PROGRAM prgMotoman
VAR
	pReal	: POINTER TO REAL;
	rVal	: REAL;
	
	pInt	: POINTER TO INT;
	iVal	: INT;
	
	fbsin	: BASIC.GEN_SIN;
	rSinOut: REAL;
	
	pRun	: POINTER TO BOOL;
	bRun	: BOOL;
	
	bUpdate: BOOL;
	
	bRunning : BOOL;
	
	fbTimer	: TOF;
	
	iCycles	: DINT;
END_VAR

pReal := ADR(GVL_io.DX200_out[0]);
//pReal^ := rVal;

pInt := ADR(GVL_io.DX200_out[4]);
//pInt^ := iVal;

pRun := ADR(GVL_io.DX200_out[0]);
pRun^ := bRun;

bRunning := GVL_io.DX200_in[0].0;

fbsin(
	PT:= T#5S, 
	AM:= 2000, 
	OS:= , 
	DL:= , 
	Q=> , 
	Out=> rSinOut);
	
IF rSinOut >= 100 THEN
	rSinOut := 100;
ELSIF rSinOut <= -100 THEN
	rSinOut := -100;
END_IF
	
IF bUpdate THEN
	pInt^ := TO_INT(rSinOut);
	iCycles := 0;
ELSE
	bRun := FALSE;
	pInt^ := 0;	
	IF bRunning THEN
		iCycles := iCycles + 1;
	END_IF
END_IF

END_PROGRAM

(* stored: Version 1.1.0.1, ProductVersion 3.1.4024.9
   POU prgMotoman: Id {795888a1-935f-43c3-9692-0fc7a23d57bd}, SpecialFunc None *)
